{region '#Template'}
	{attribute 'Version' := '5.0.0.0'}
	{attribute 'Tags' := '"LCID": "1031", "Text": "AC, Aggregates, ERC, Plate"'}
	{attribute 'Tags' := '"LCID": "1033", "Text": "AC, Aggregates, ERC, Plate"'}
	{attribute 'Using' := '"Type": "Template", "URI": "BA2_Param"'}
	{attribute 'Using' := '"Type": "Template", "URI": "EC_ID"'}
	{attribute 'Description' := '"LCID": "1031", "Text": "Aggregat Energie Rückgewinnung Platte mit Bypass"'}
	{attribute 'Description' := '"LCID": "1033", "Text": "Aggregate energy recovery plate with bypass"'}
{endregion}
FUNCTION_BLOCK FB_BA_AC_ErcPl_02 EXTENDS FB_BA_View
VAR_INPUT
	fSpTSuA					: REAL;
	fTSuA					: REAL;
	bSyncTSuACtrl			: BOOL;
	fSyncTSuACtrl			: REAL;			
	bDehumf					: BOOL;
	fTExhA					: REAL;
	fTExtA					: REAL;
	fTWth					: REAL;
	stCmd					: ST_BA_Binary;				
END_VAR
VAR_OUTPUT
	fPresentValue			: REAL;				
	eAction					: E_BA_Action;
	bActiveSeqCtrl			: BOOL;	
END_VAR
VAR_IN_OUT
	stTSeqLink				: ST_BA_SeqLink;	//	Sequenz Link Struktur	//	Sequence link structure	
END_VAR
VAR_INPUT CONSTANT
	TSuACtrl				: FB_BA_AC_ErcTSuACtrl;								 
	TExhACtrl				: FB_BA_PID_Sp;		
	DiffPrssSwi				: FB_BA_SensorBinary_Raw;							
	IcePrtcRamp				: FB_BA_RampLimitIncrease;								
	Dmp						: FB_BA_ActuatorAnalog;
	ByDmp					: FB_BA_ActuatorAnalog;					
	PlantLock				: FB_BA_PlantLock;		
END_VAR
VAR
	bPrioSfty				: BOOL;
	bPrioCrit				: BOOL;		
	PrioSwiVal				: FB_BA_PrioSwi_B04;	
	Inv						: FB_BA_Chrct02;	
END_VAR
VAR // added by the converter: edge detectors and wires of the graphical bodies
    _s1, _s2 : ST_BA_Analog;
    _w1 : ANY;
END_VAR

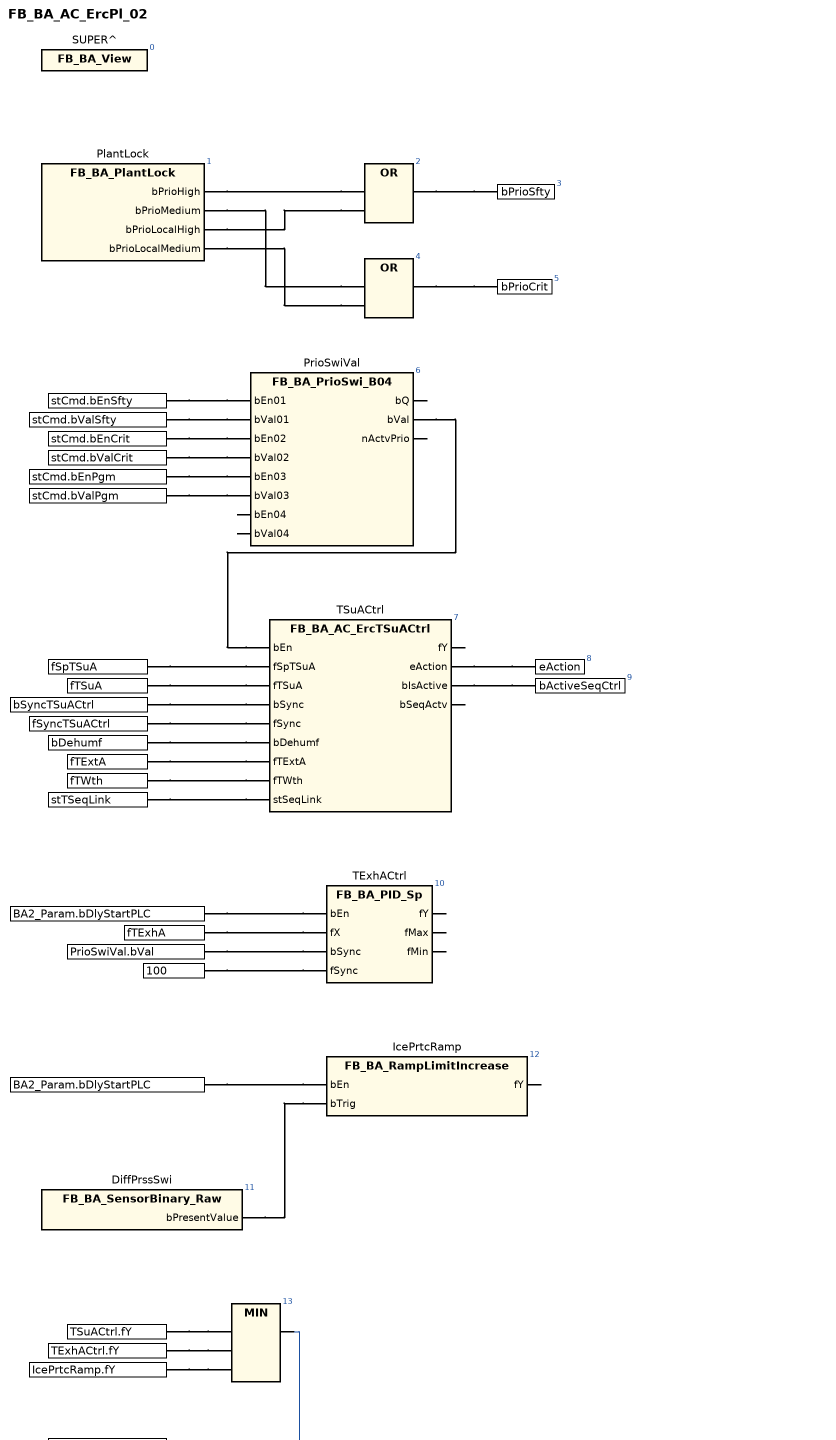
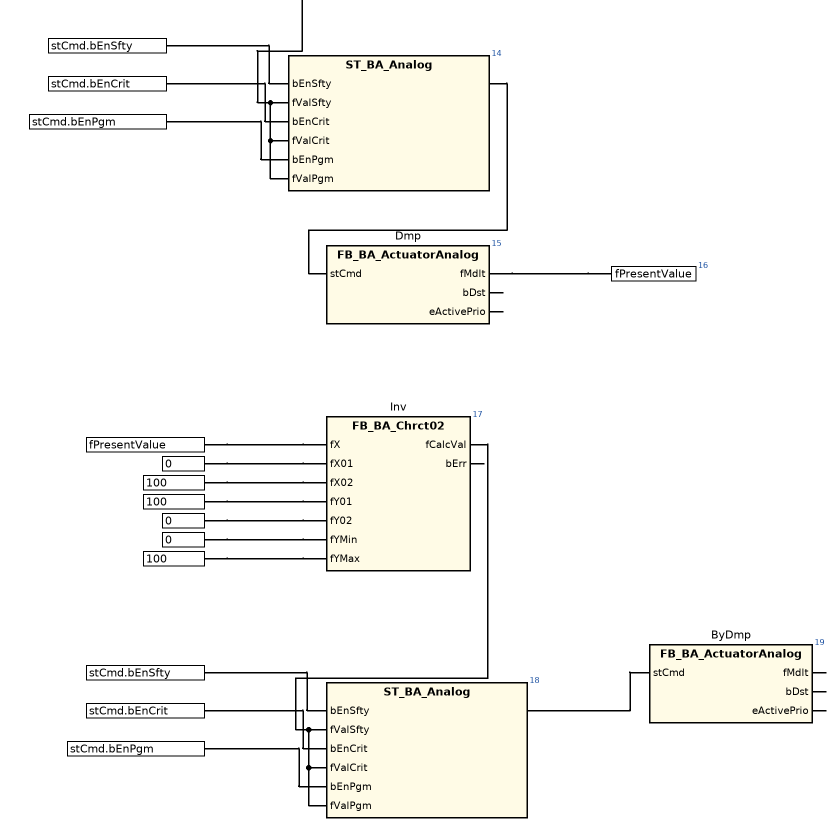
SUPER^(); // FB_BA_View
PlantLock(); // FB_BA_PlantLock
bPrioSfty := PlantLock.bPrioHigh OR PlantLock.bPrioLocalHigh;
bPrioCrit := PlantLock.bPrioMedium OR PlantLock.bPrioLocalMedium;
PrioSwiVal(
    bEn01 := stCmd.bEnSfty,
    bVal01 := stCmd.bValSfty,
    bEn02 := stCmd.bEnCrit,
    bVal02 := stCmd.bValCrit,
    bEn03 := stCmd.bEnPgm,
    bVal03 := stCmd.bValPgm); // FB_BA_PrioSwi_B04
TSuACtrl(
    bEn := PrioSwiVal.bVal,
    fSpTSuA := fSpTSuA,
    fTSuA := fTSuA,
    bSync := bSyncTSuACtrl,
    fSync := fSyncTSuACtrl,
    bDehumf := bDehumf,
    fTExtA := fTExtA,
    fTWth := fTWth,
    stSeqLink := stTSeqLink); // FB_BA_AC_ErcTSuACtrl
eAction := TSuACtrl.eAction;
bActiveSeqCtrl := TSuACtrl.bIsActive;
TExhACtrl(bEn := BA2_Param.bDlyStartPLC, fX := fTExhA, bSync := PrioSwiVal.bVal, fSync := 100); // FB_BA_PID_Sp
DiffPrssSwi(); // FB_BA_SensorBinary_Raw
IcePrtcRamp(bEn := BA2_Param.bDlyStartPLC, bTrig := DiffPrssSwi.bPresentValue); // FB_BA_RampLimitIncrease
_w1 := MIN(TSuACtrl.fY, TExhACtrl.fY, IcePrtcRamp.fY);
// compose _s1 : ST_BA_Analog
_s1.bEnSfty := stCmd.bEnSfty;
_s1.fValSfty := _w1;
_s1.bEnCrit := stCmd.bEnCrit;
_s1.fValCrit := _w1;
_s1.bEnPgm := stCmd.bEnPgm;
_s1.fValPgm := _w1;
Dmp(stCmd := _s1); // FB_BA_ActuatorAnalog
fPresentValue := Dmp.fMdlt;
Inv(fX := fPresentValue, fX01 := 0, fX02 := 100, fY01 := 100, fY02 := 0, fYMin := 0, fYMax := 100); // FB_BA_Chrct02
// compose _s2 : ST_BA_Analog
_s2.bEnSfty := stCmd.bEnSfty;
_s2.fValSfty := Inv.fCalcVal;
_s2.bEnCrit := stCmd.bEnCrit;
_s2.fValCrit := Inv.fCalcVal;
_s2.bEnPgm := stCmd.bEnPgm;
_s2.fValPgm := Inv.fCalcVal;
ByDmp(stCmd := _s2); // FB_BA_ActuatorAnalog

METHOD FB_init : BOOL
VAR_INPUT
	bInitRetains : BOOL; // if TRUE, the retain variables are initialized (warm start / cold start)
	bInCopyCode : BOOL;  // if TRUE, the instance afterwards gets moved into the copy code (online change)
END_VAR
PlantLock.Parent								:= THIS^;		

TSuACtrl.iParent								:= THIS^;	 
TSuACtrl.iLabel									:= LblCtl_SupplyAirTemperatureControl;   
TSuACtrl.sObjectName							:= '{Idx=21}';						 
TSuACtrl.eDPADMode								:= E_BA_DPADMode.eInclude;								

TExhACtrl.iParent								:= THIS^;	
TExhACtrl.iLabel								:= LblCtl_ExhaustAirTemperatureControl;  
TExhACtrl.sObjectName							:= '{Idx=22}';						 
TExhACtrl.eDPADMode								:= E_BA_DPADMode.eInclude;	
TExhACtrl.Sp.fValueRm 							:= 3.0;
TExhACtrl.Ctrl.eActionRm						:= E_BA_Action.eDirect;			

DiffPrssSwi.iParent								:= THIS^;	
DiffPrssSwi.iLabel								:= LblAgg_PressureDifferential;  
DiffPrssSwi.sObjectName							:= '{Idx=21}';						 
DiffPrssSwi.eDPADMode							:= E_BA_DPADMode.eInclude;
DiffPrssSwi.Input.iLabel						:= LblFun_OperationalMessage;   
DiffPrssSwi.Input.sObjectName					:= '{Idx=01}';						 
DiffPrssSwi.Input.ePolarity						:= E_BA_Polarity.eReverse;
DiffPrssSwi.Input.sActiveText 					:= txtEvent_Triggered;
DiffPrssSwi.Input.sInactiveText 				:= txtEvent_Normal;
DiffPrssSwi.Input.nEventClassID					:= EC_ID.NC30;
DiffPrssSwi.Input.aEventTransitionText[1]		:= txtEvent_Triggered;
DiffPrssSwi.Input.aEventTransitionText[2]		:= txtEvent_Error;
DiffPrssSwi.Input.aEventTransitionText[3]		:= txtEvent_Normal;
DiffPrssSwi.Input.bEventDetectionEnable			:= TRUE;
DiffPrssSwi.Input.eEnPlantLock					:= E_BA_LockPriority.eNoLock;	


IcePrtcRamp.iParent								:= THIS^;	
IcePrtcRamp.iLabel								:= LblCtl_EnergyRecoveryDeicingRamp;   
IcePrtcRamp.sObjectName							:= '{Idx=21}';						 
IcePrtcRamp.eDPADMode							:= E_BA_DPADMode.eIncludeDescription;
IcePrtcRamp.TiUp.fValueRm						:= 1200;

Dmp.iParent										:= THIS^;
Dmp.iLabel										:= LblAgg_VentilationDamperSupplyAir;   										 
Dmp.sObjectName									:= '{Idx=21}';						 
Dmp.eDPADMode									:= E_BA_DPADMode.eInclude;
Dmp.Mdlt.fResolution 							:= 0.003814755;
Dmp.Mdlt.fScaleOffset 							:= 0;

ByDmp.iParent									:= THIS^;
ByDmp.iLabel									:= LblAgg_VentilationDamperBypassAir;   									 
ByDmp.sObjectName								:= '{Idx=22}';						 
ByDmp.eDPADMode									:= E_BA_DPADMode.eInclude;
ByDmp.Mdlt.fResolution 							:= 0.003814755;
ByDmp.Mdlt.fScaleOffset 						:= 0;
END_METHOD

END_FUNCTION_BLOCK

(* stored: Version 1.1.0.1, ProductVersion 3.1.4024.12
   POU FB_BA_AC_ErcPl_02: Id {e7b824ec-3312-4911-854f-4f41635859bf}, SpecialFunc None
   Method FB_init: Id {443efafb-1b45-48fb-ac7d-5e0cab38e44a} *)
